Staubli VAL3: SpeedFilter.pgx

public program SpeedFilter(trsf x_tr, mdesc& x_mDest)
  local num l_nDist
begin

 // DataBase:nSpeedPercent=min(max(0.001,DataBase:nSpeedPercent),100)



  //调试系数
  //l_nPercent=2
  //








  x_mDest.decel=x_mDest.accel=max(x_tr.rx,0.1)*1
  x_mDest.blend=Cartesian
   // x_mDest.blend=joint
  x_mDest.reach=x_mDest.leave=max(x_tr.ry,0)
  x_mDest.tvel=max(x_tr.z,0.1)*1
  x_mDest.vel=100
  x_mDest.rvel=99999


end
